FUNCTION F_DWORD_RTN : DWORD
VAR_INPUT
	stArg : ST_Arg;
END_VAR
VAR
	sysVar_Info : __SYSTEM.VAR_INFO;
END_VAR

sysVar_Info := __VARINFO(F_DWORD_RTN);
IF stArg.TypeClass = sysVar_Info.TypeClass THEN 
	F_DWORD_RTN := TO_DWORD(stArg.sValue);
	END_IF

END_FUNCTION

(* stored: Version 1.1.0.1, ProductVersion 3.1.4024.4
   POU F_DWORD_RTN: Id {d86f7841-64f2-4ccc-9842-29458f20dc7d}, SpecialFunc None *)
